// LS Electric XG5000 project: ASCII_Slave_last
// PLC LSPLC

PROGRAM 50_SerialComm (task: 스캔 프로그램)

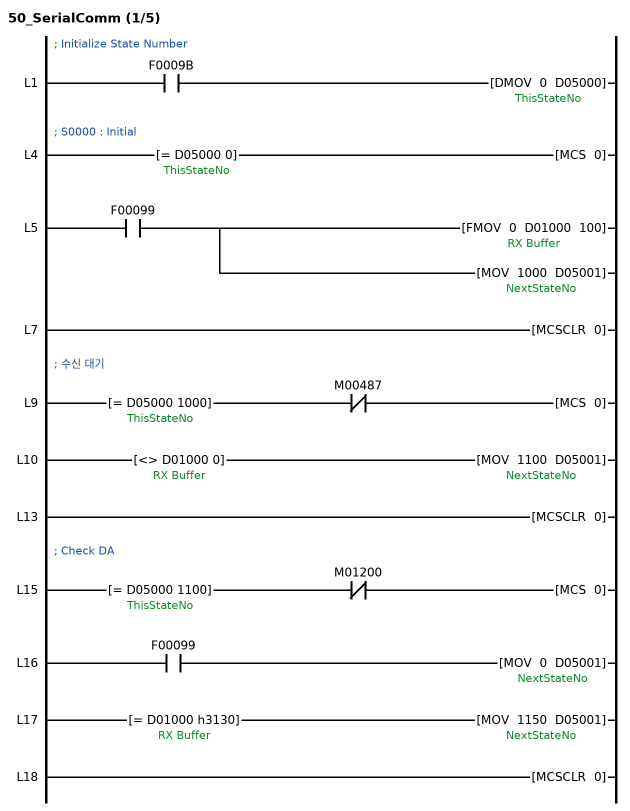
// Initialize State Number
; L1
LOAD      F0009B
DMOV      0 D05000	// ThisStateNo
// S0000 : Initial
; L4
LOAD=     D05000 0	// ThisStateNo
MCS       0
; L5
LOAD      F00099
FMOV      0 D01000 100	// RX Buffer
MOV       1000 D05001	// NextStateNo
; L7
MCSCLR    0
// 수신 대기
; L9
LOAD=     D05000 1000	// ThisStateNo
AND NOT   M00487
MCS       0
; L10
LOAD<>    D01000 0	// RX Buffer
MOV       1100 D05001	// NextStateNo
; L13
MCSCLR    0
// Check DA
; L15
LOAD=     D05000 1100	// ThisStateNo
AND NOT   M01200
MCS       0
; L16
LOAD      F00099
MOV       0 D05001	// NextStateNo
; L17
LOAD=     D01000 h3130	// RX Buffer
MOV       1150 D05001	// NextStateNo
; L18
MCSCLR    0

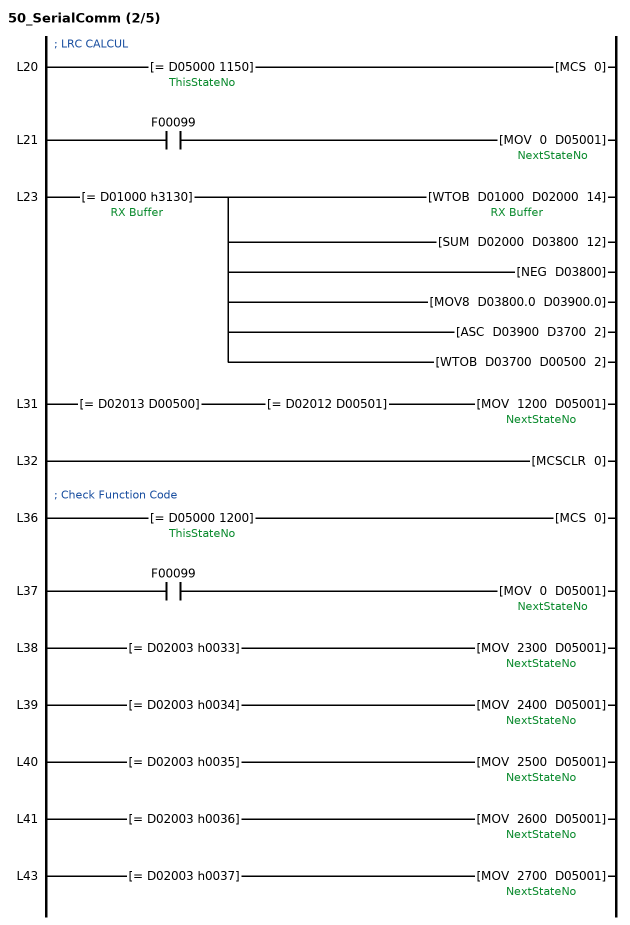
// LRC CALCUL
; L20
LOAD=     D05000 1150	// ThisStateNo
MCS       0
; L21
LOAD      F00099
MOV       0 D05001	// NextStateNo
; L23
LOAD=     D01000 h3130	// RX Buffer
WTOB      D01000 D02000 14	// RX Buffer
SUM       D02000 D03800 12
NEG       D03800
MOV8      D03800.0 D03900.0
ASC       D03900 D3700 2
WTOB      D03700 D00500 2
; L31
LOAD=     D02013 D00500
AND=      D02012 D00501
MOV       1200 D05001	// NextStateNo
; L32
MCSCLR    0
// Check Function Code
; L36
LOAD=     D05000 1200	// ThisStateNo
MCS       0
; L37
LOAD      F00099
MOV       0 D05001	// NextStateNo
; L38
LOAD=     D02003 h0033
MOV       2300 D05001	// NextStateNo
; L39
LOAD=     D02003 h0034
MOV       2400 D05001	// NextStateNo
; L40
LOAD=     D02003 h0035
MOV       2500 D05001	// NextStateNo
; L41
LOAD=     D02003 h0036
MOV       2600 D05001	// NextStateNo
; L43
LOAD=     D02003 h0037
MOV       2700 D05001	// NextStateNo

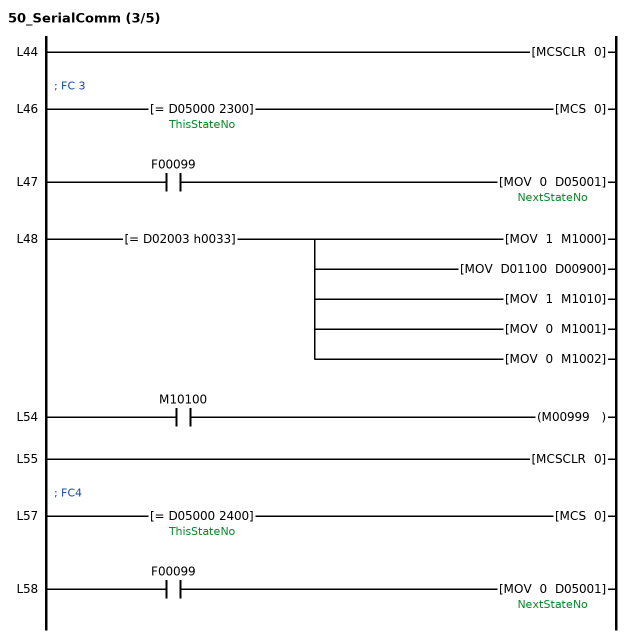
; L44
MCSCLR    0
// FC 3
; L46
LOAD=     D05000 2300	// ThisStateNo
MCS       0
; L47
LOAD      F00099
MOV       0 D05001	// NextStateNo
; L48
LOAD=     D02003 h0033
MOV       1 M1000
MOV       D01100 D00900
MOV       1 M1010
MOV       0 M1001
MOV       0 M1002
; L54
LOAD      M10100
OUT       M00999
; L55
MCSCLR    0
// FC4
; L57
LOAD=     D05000 2400	// ThisStateNo
MCS       0
; L58
LOAD      F00099
MOV       0 D05001	// NextStateNo

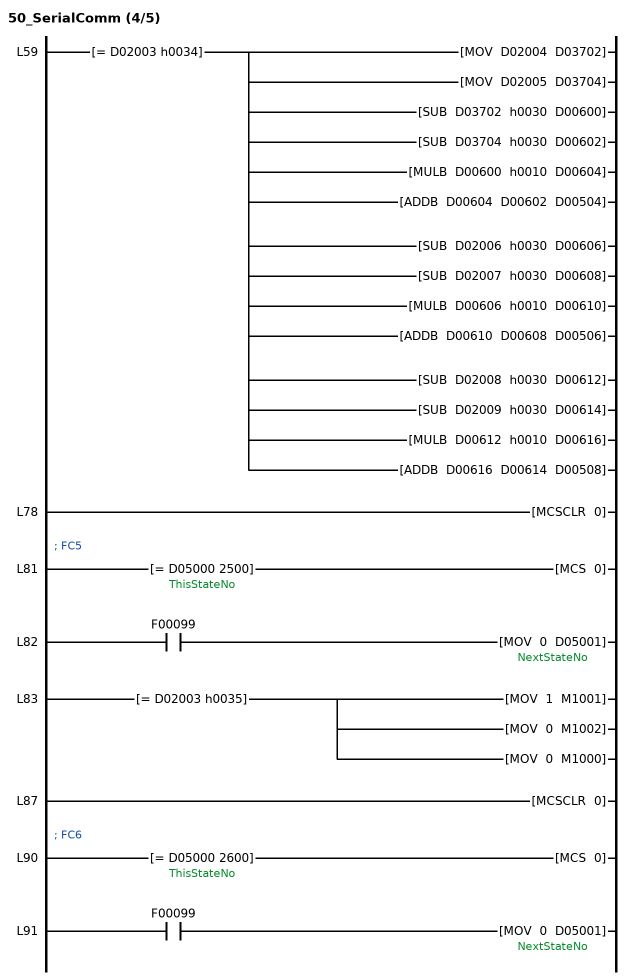
; L59
LOAD=     D02003 h0034
MOV       D02004 D03702
MOV       D02005 D03704
SUB       D03702 h0030 D00600
SUB       D03704 h0030 D00602
MULB      D00600 h0010 D00604
ADDB      D00604 D00602 D00504
SUB       D02006 h0030 D00606
SUB       D02007 h0030 D00608
MULB      D00606 h0010 D00610
ADDB      D00610 D00608 D00506
SUB       D02008 h0030 D00612
SUB       D02009 h0030 D00614
MULB      D00612 h0010 D00616
ADDB      D00616 D00614 D00508
; L78
MCSCLR    0
// FC5
; L81
LOAD=     D05000 2500	// ThisStateNo
MCS       0
; L82
LOAD      F00099
MOV       0 D05001	// NextStateNo
; L83
LOAD=     D02003 h0035
MOV       1 M1001
MOV       0 M1002
MOV       0 M1000
; L87
MCSCLR    0
// FC6
; L90
LOAD=     D05000 2600	// ThisStateNo
MCS       0
; L91
LOAD      F00099
MOV       0 D05001	// NextStateNo

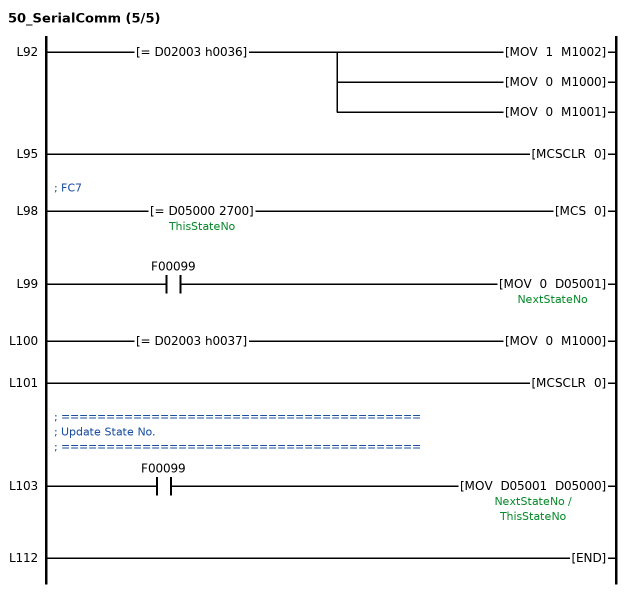
; L92
LOAD=     D02003 h0036
MOV       1 M1002
MOV       0 M1000
MOV       0 M1001
; L95
MCSCLR    0
// FC7
; L98
LOAD=     D05000 2700	// ThisStateNo
MCS       0
; L99
LOAD      F00099
MOV       0 D05001	// NextStateNo
; L100
LOAD=     D02003 h0037
MOV       0 M1000
; L101
MCSCLR    0
// ========================================
// Update State No.
// ========================================
; L103
LOAD      F00099
MOV       D05001 D05000	// NextStateNo / ThisStateNo
; L112
END

PROGRAM 60_TX_Flag (task: 스캔 프로그램)

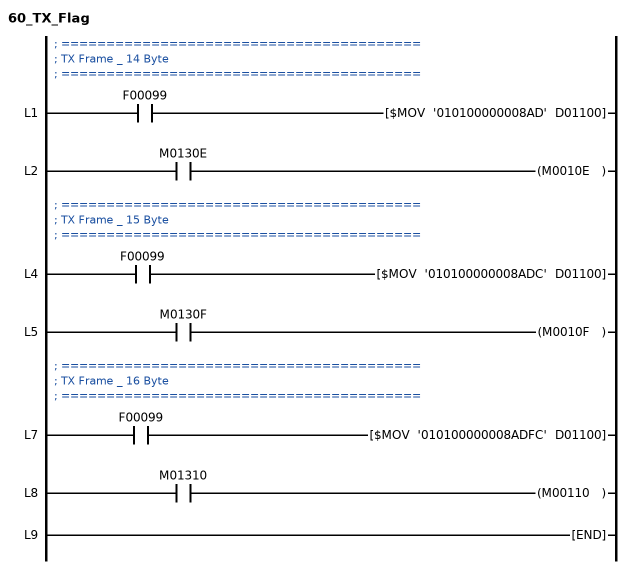
// ========================================
// TX Frame _ 14 Byte
// ========================================
; L1
LOAD      F00099
$MOV      '010100000008AD' D01100
; L2
LOAD      M0130E
OUT       M0010E
// ========================================
// TX Frame _ 15 Byte
// ========================================
; L4
LOAD      F00099
$MOV      '010100000008ADC' D01100
; L5
LOAD      M0130F
OUT       M0010F
// ========================================
// TX Frame _ 16 Byte
// ========================================
; L7
LOAD      F00099
$MOV      '010100000008ADFC' D01100
; L8
LOAD      M01310
OUT       M00110
; L9
END

PROGRAM convey (task: 스캔 프로그램)

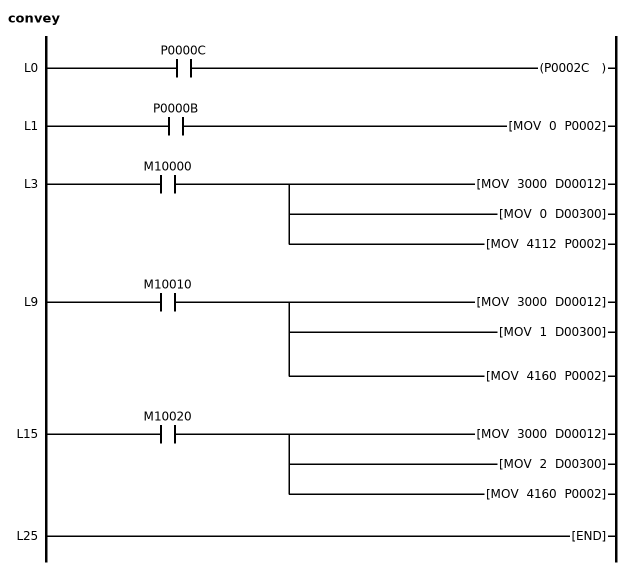
; L0
LOAD      P0000C
OUT       P0002C
; L1
LOAD      P0000B
MOV       0 P0002
; L3
LOAD      M10000
MOV       3000 D00012
MOV       0 D00300
MOV       4112 P0002
; L9
LOAD      M10010
MOV       3000 D00012
MOV       1 D00300
MOV       4160 P0002
; L15
LOAD      M10020
MOV       3000 D00012
MOV       2 D00300
MOV       4160 P0002
; L25
END

PROGRAM tp_inter (task: 스캔 프로그램)

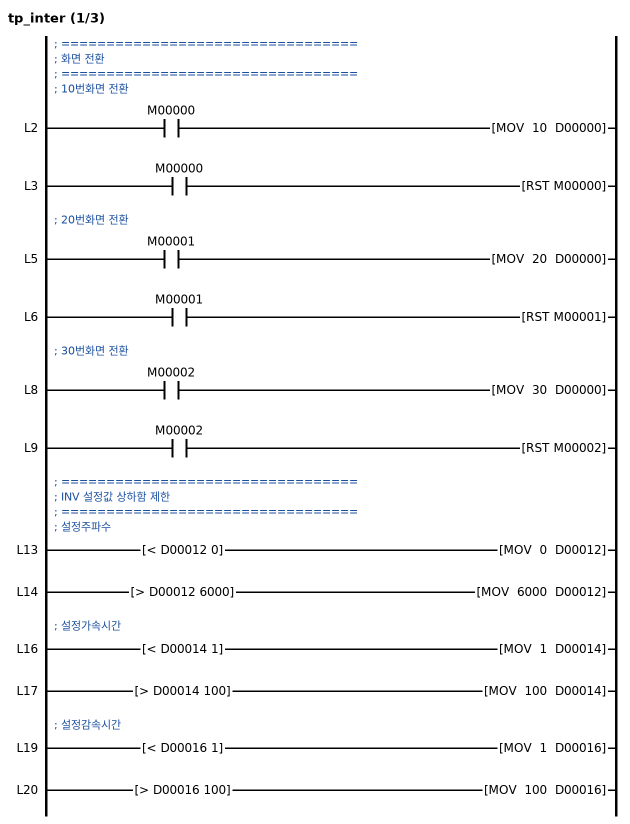
// =================================
//    화면 전환
// =================================
// 10번화면 전환
; L2
LOAD      M00000
MOV       10 D00000
; L3
LOAD      M00000
RST       M00000
// 20번화면 전환
; L5
LOAD      M00001
MOV       20 D00000
; L6
LOAD      M00001
RST       M00001
// 30번화면 전환
; L8
LOAD      M00002
MOV       30 D00000
; L9
LOAD      M00002
RST       M00002
// =================================
//    INV 설정값 상하함 제한
// =================================
// 설정주파수
; L13
LOAD<     D00012 0
MOV       0 D00012
; L14
LOAD>     D00012 6000
MOV       6000 D00012
// 설정가속시간
; L16
LOAD<     D00014 1
MOV       1 D00014
; L17
LOAD>     D00014 100
MOV       100 D00014
// 설정감속시간
; L19
LOAD<     D00016 1
MOV       1 D00016
; L20
LOAD>     D00016 100
MOV       100 D00016

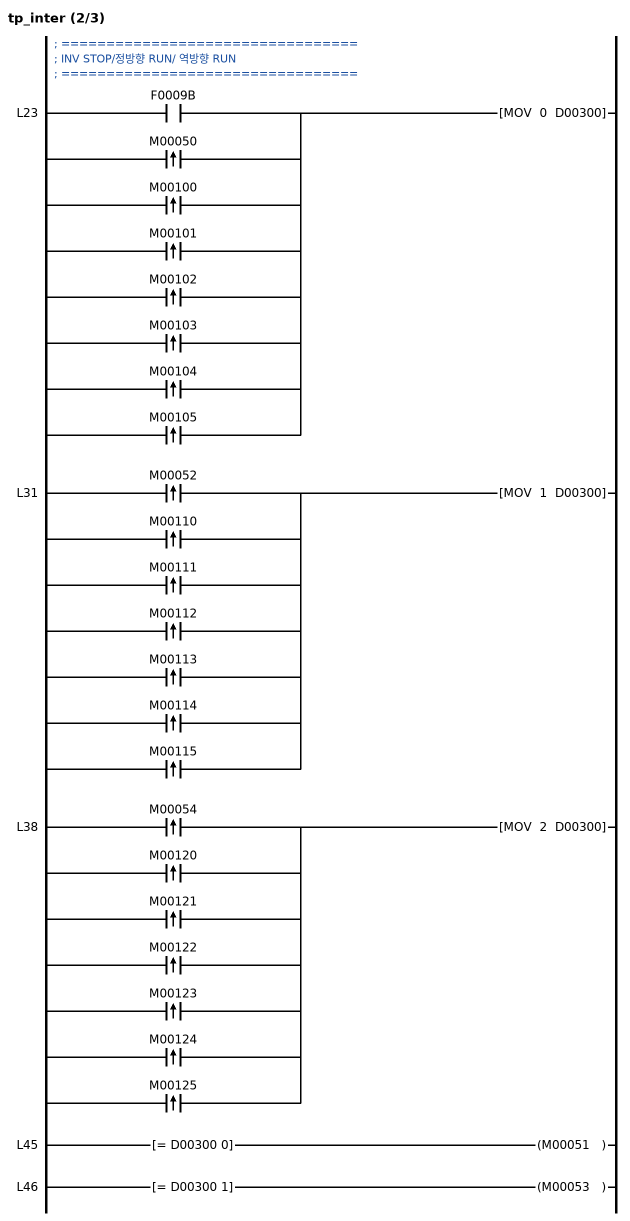
// =================================
//    INV STOP/정방향 RUN/ 역방향 RUN
// =================================
; L23
LOAD      F0009B
ORP       M00050
ORP       M00100
ORP       M00101
ORP       M00102
ORP       M00103
ORP       M00104
ORP       M00105
MOV       0 D00300
; L31
LOADP     M00052
ORP       M00110
ORP       M00111
ORP       M00112
ORP       M00113
ORP       M00114
ORP       M00115
MOV       1 D00300
; L38
LOADP     M00054
ORP       M00120
ORP       M00121
ORP       M00122
ORP       M00123
ORP       M00124
ORP       M00125
MOV       2 D00300
; L45
LOAD=     D00300 0
OUT       M00051
; L46
LOAD=     D00300 1
OUT       M00053

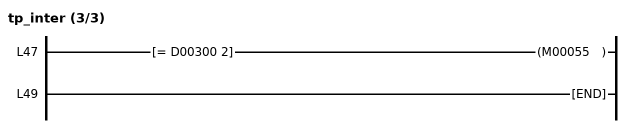
; L47
LOAD=     D00300 2
OUT       M00055
; L49
END

PROGRAM inv (task: 스캔 프로그램)

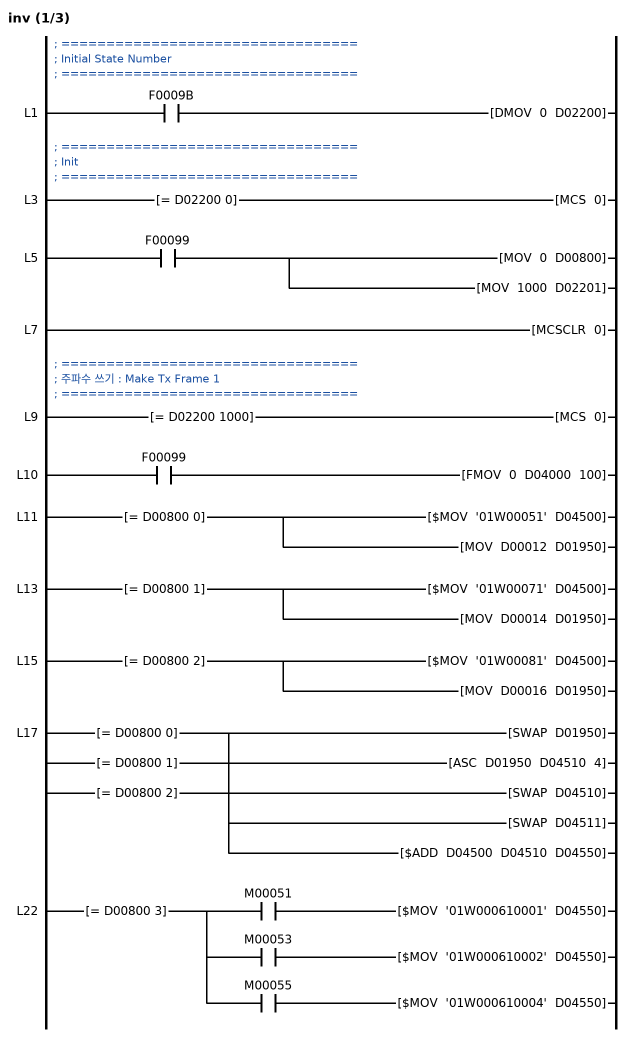
// =================================
//    Initial State Number
// =================================
; L1
LOAD      F0009B
DMOV      0 D02200
// =================================
//    Init
// =================================
; L3
LOAD=     D02200 0
MCS       0
; L5
LOAD      F00099
MOV       0 D00800
MOV       1000 D02201
; L7
MCSCLR    0
// =================================
//    주파수 쓰기 : Make Tx Frame 1
// =================================
; L9
LOAD=     D02200 1000
MCS       0
; L10
LOAD      F00099
FMOV      0 D04000 100
; L11
LOAD=     D00800 0
$MOV      '01W00051' D04500
MOV       D00012 D01950
; L13
LOAD=     D00800 1
$MOV      '01W00071' D04500
MOV       D00014 D01950
; L15
LOAD=     D00800 2
$MOV      '01W00081' D04500
MOV       D00016 D01950
; L17
LOAD=     D00800 0
OR=       D00800 1
OR=       D00800 2
SWAP      D01950
ASC       D01950 D04510 4
SWAP      D04510
SWAP      D04511
$ADD      D04500 D04510 D04550
; L22
LOAD=     D00800 3
MPUSH
AND       M00051
$MOV      '01W000610001' D04550
MLOAD
AND       M00053
$MOV      '01W000610002' D04550
MPOP
AND       M00055
$MOV      '01W000610004' D04550

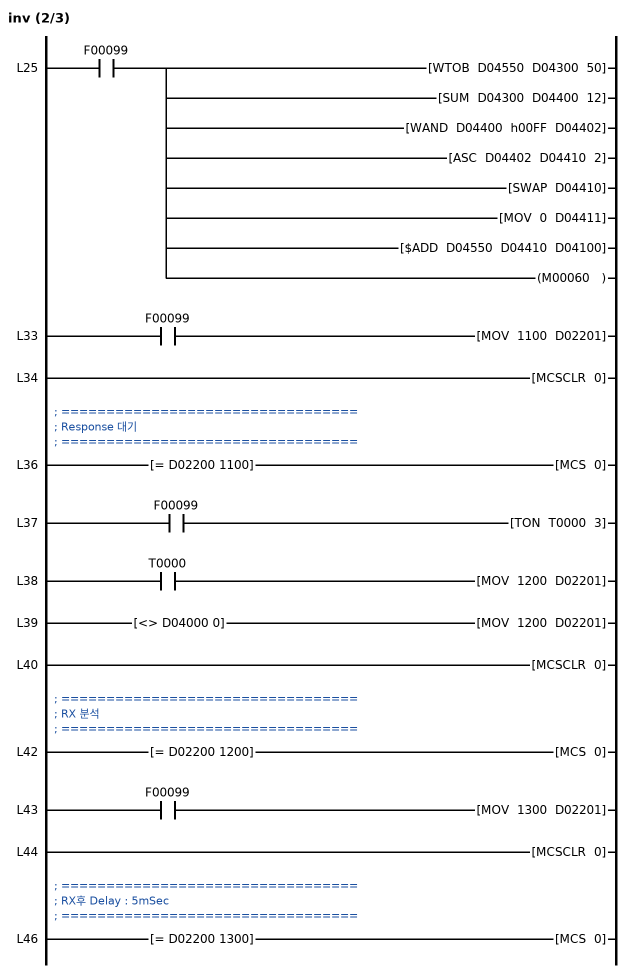
; L25
LOAD      F00099
WTOB      D04550 D04300 50
SUM       D04300 D04400 12
WAND      D04400 h00FF D04402
ASC       D04402 D04410 2
SWAP      D04410
MOV       0 D04411
$ADD      D04550 D04410 D04100
OUT       M00060
; L33
LOAD      F00099
MOV       1100 D02201
; L34
MCSCLR    0
// =================================
//    Response 대기
// =================================
; L36
LOAD=     D02200 1100
MCS       0
; L37
LOAD      F00099
TON       T0000 3
; L38
LOAD      T0000
MOV       1200 D02201
; L39
LOAD<>    D04000 0
MOV       1200 D02201
; L40
MCSCLR    0
// =================================
//    RX 분석
// =================================
; L42
LOAD=     D02200 1200
MCS       0
; L43
LOAD      F00099
MOV       1300 D02201
; L44
MCSCLR    0
// =================================
//    RX후 Delay : 5mSec
// =================================
; L46
LOAD=     D02200 1300
MCS       0

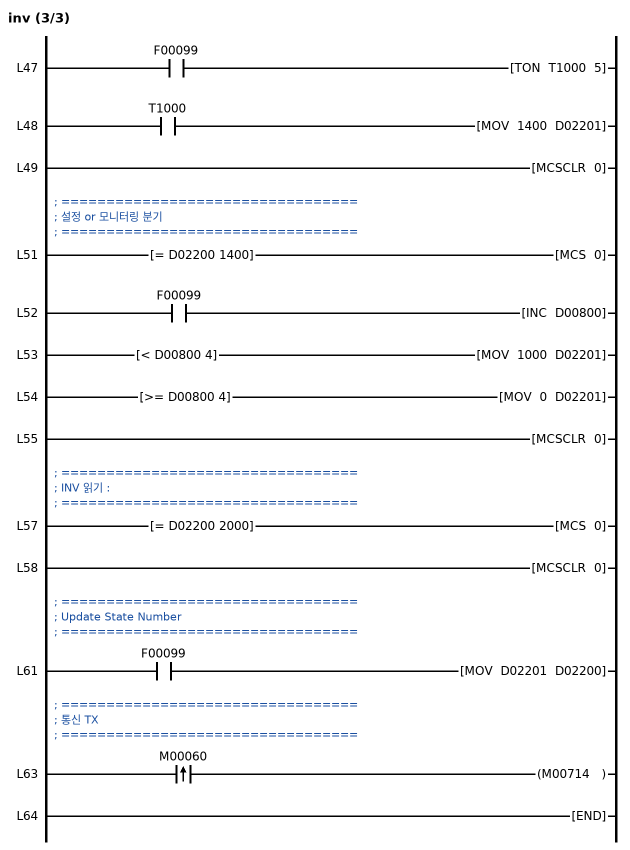
; L47
LOAD      F00099
TON       T1000 5
; L48
LOAD      T1000
MOV       1400 D02201
; L49
MCSCLR    0
// =================================
//    설정 or 모니터링 분기
// =================================
; L51
LOAD=     D02200 1400
MCS       0
; L52
LOAD      F00099
INC       D00800
; L53
LOAD<     D00800 4
MOV       1000 D02201
; L54
LOAD>=    D00800 4
MOV       0 D02201
; L55
MCSCLR    0
// =================================
//    INV 읽기 :
// =================================
; L57
LOAD=     D02200 2000
MCS       0
; L58
MCSCLR    0
// =================================
//    Update State Number
// =================================
; L61
LOAD      F00099
MOV       D02201 D02200
// =================================
//    통신 TX
// =================================
; L63
LOADP     M00060
OUT       M00714
; L64
END

VARIABLES AND COMMENTS (devices not used above)
D02001	WORD	RX Function Code
D03500	WORD	연산 CRC
D03562	WORD	수신 CRC
D03560	WORD	CRC 연산할 Byte 수
M00106	BIT	TxFlag for Read Coil Status